FUNCTION_BLOCK SpringCyl (* Basic Function Block Type *)
  (* Standard: 61499-2 *)
  (* Version 0.2, 2003-12-04, JHC, Rockwell Automation, Renamed for better indexing. *)
  (* Version 0.1, 2002-11-05, JHC, Rockwell Automation, Corrected missing ST element in Algorithm REQ. *)
  (* Version 0.0, 2000-05-30, JHC, Rockwell Automation *)
  (* Compiler header: package fb.rt.pnp; *)
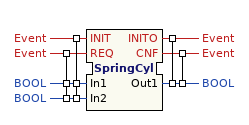
  EVENT_INPUT
    INIT WITH In1, In2; (* Initialization Request *)
    REQ WITH In1, In2; (* Normal Execution Request *)
  END_EVENT
  EVENT_OUTPUT
    INITO WITH Out1; (* Initialization Confirm *)
    CNF WITH Out1; (* Execution Confirmation *)
  END_EVENT
  VAR_INPUT
    In1 : BOOL; (* Input event qualifier *)
    In2 : BOOL;
  END_VAR
  VAR_OUTPUT
    Out1 : BOOL; (* Output event qualifier *)
  END_VAR
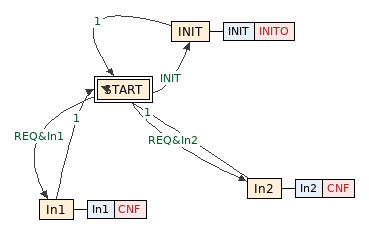
  EC_STATES
    START; (* Initial State *)
    INIT : INIT -> INITO; (* Initialization *)
    In1 : In1 -> CNF; (* Normal execution *)
    In2 : In2 -> CNF;
  END_STATES
  EC_TRANSITIONS
    START TO INIT := INIT;
    INIT TO START := 1;
    START TO In1 := REQ&In1;
    In1 TO START := 1;
    START TO In2 := REQ&In2;
    In2 TO START := 1;
  END_TRANSITIONS
  ALGORITHM INIT IN ST: (* Initialization algorithm *)

  END_ALGORITHM
  ALGORITHM In1 IN ST: (* Normally executed algorithm *)
Out1 := In1;
System.out.println("In1!!!!");
  END_ALGORITHM
  ALGORITHM In2 IN ST: (* Normally executed algorithm *)
Out1:=In1;
System.out.println("In2!!!!" + Out1);
  END_ALGORITHM
END_FUNCTION_BLOCK
